{attribute addProperty BoxType "EKM1101-0000-0016"}
{attribute addProperty Id "TimestampAT %I*ULINT648"}
{attribute addProperty CRC "187023780"}
{attribute addProperty SizeInBites "64"}
{attribute addProperty SizeInBytes "8"}
TYPE MMS_Acceleration_Timestamp_0B25C1A4 :
STRUCT
	{attribute addProperty Name "Timestamp"}
	Timestamp AT %I* : ULINT;
END_STRUCT
END_TYPE

(* stored: Version 1.2.0.0, ProductVersion 3.1.4024.9
   DUT MMS_Acceleration_Timestamp_0B25C1A4: Id {636efea0-4798-42fa-9031-45ad1db1d893} *)
